(* PLC project Tc3_EventLogger.ExtendName Demo, tc3-libraries-kb TwinCAT 3.1 *)
(* stored: creationDateTime 2026-05-11T01:00:00, modificationDateTime 2026-05-11T01:00:00 *)

PROGRAM P_Demo_ExtendName
  VAR
    fbSrc : FB_TcSourceInfo;  (* 源信息实例 *)
    sStationId : STRING := 'Station-01';  (* 工位号后缀 *)
    bDoExtend : BOOL := FALSE;  (* 上升沿触发 *)
    bDoExtendPrev : BOOL;  (* 边沿检测 *)
    hr : HRESULT;  (* 返回值监视 *)
  END_VAR

// =============================================================================
// 场景：给当前工位的 SourceInfo 加工位号后缀
// 价值：事件天然带工位标识
// 验证：登录后调用一次 ExtendName 后 fbSrc.sSourceName 应包含 sExtName 内容
// 验证步骤：
//   1. 右键 PLC 项目 → Import PLCopenXML → 选本文件
//   2. 引用 Tc3_EventLogger（System → References → Add library）
//   3. 编译 → 登录 → 运行；按 verify 注释里给出的在线写值操作
// =============================================================================

IF bDoExtend AND NOT bDoExtendPrev THEN
    hr := fbSrc.ExtendName(sExtName := sStationId);
END_IF;
bDoExtendPrev := bDoExtend;
END_PROGRAM
